DATA_BLOCK "dbArchiveAutoOven"
{ S7_Optimized_Access := 'TRUE' }
VERSION : 0.8
NON_RETAIN
"fbArchiveAutoOven"

BEGIN

END_DATA_BLOCK

